Universal Robots PolyScope program: Force to distance.urp

Program Force to distance (installation=default directory=/programs createdIn=5.10.0.106268 lastSavedIn=5.10.0.106268 robotSerialNumber=20185500191)
Calibrated DH parameters: a=[0.000131, -0.165639, -0.102041, 0.000082, 0.000046, 0]; d=[0.162455, 220.258006, 1988.136334, -2208.260978, 0.099826, 0.099896]; alpha=[1.570482, -0.001777, -0.000172, 1.570393, -1.570735, 0]; deltaTheta=[0, -1.170526, -0.137148, 1.307669, -0.000001, 0]
BeforeStart
  Travel_Distance := 0.25
  Time_out := 5
  Distance_pose := p[0,0,0,0,0,0]
  forceEvent := False
  forceComplete := False
Robot Program (runOnlyOnce=false)
  MoveJ speed 60 deg/s, acceleration 80 deg/s^2 (useActiveTCP=true) feature=Base
    Waypoint Approach: TCP in base x=246.187 y=-360.171 z=399.264 mm, rx=-2.1879 ry=-2.2382 rz=-0.0171 rad; joints [-38.302, -81.57, -84.97, -104.059, 90.62, 140.416] deg; TCP offset x=0 y=0 z=174 mm, rx=0 ry=0 rz=0 rad
    Waypoint Force_Start: TCP in base x=449.999 y=-365.041 z=133.455 mm, rx=-2.188 ry=-2.2544 rz=0 rad; joints [-25.743, -104.782, -100.25, -64.972, 89.919, 152.525] deg
  'This loop just makes sure the robot is fully at rest before taring.'
  Loop While (checkContinuously=false) expression=is_steady()≟ False
    Script: is_steady()
    Script: sync()
  Cur_Pose := get_actual_tcp_pose()
  Script: zero_ftsensor()
  Timer (action=Start) variable(name=timer_1)
  forceEvent := True
  Force Frame feature=Base; selection=[1, 1, 1, 0, 0, 0]; wrench=[0, -15, 0, 0, 0, 0]; limitsForce=[0.005, 0.1, 0.005, 1.047198, 1.047198, 1.047198]; limitsMotion=[0.1, 0.1, 0.1, 0.349066, 0.349066, 0.349066]
    Wait Condition expression=forceComplete≟ True
  Script: stopl(2)
  forceComplete := False
  Timer (action=Stop) variable=timer_1
  If timer_1>Time_out
    Popup Error (haltProgram=false message=Distance not reached! inputType=Text)
    Timer (action=Reset) variable=timer_1
    Halt
  Timer (action=Reset) variable=timer_1
Event  expression=forceEvent≟ True
  Force_Pose := get_actual_tcp_pose()
  Distance_pose := pose_sub(Cur_Pose, Force_Pose)
  If timer_1>Time_out or Distance_pose[0]>Travel_Distance
    forceComplete := True
    Distance_pose := p[0,0,0,0,0,0]
    forceEvent := False
  Script: sync()
